// TIA Portal V19 export
TYPE "typePressureGuageRs485ControlNodeMonitoring"
TITLE = LBC_typeAnalogOutputControlNodeMonitoring
// Control Node Wapper monitoring values
// stored: Access Published
   STRUCT
      valid { ExternalAccessible := 'False'; ExternalVisible := 'False'; ExternalWritable := 'False'} : Bool;   // Manual mode parameters for axis control interface
      busy { ExternalAccessible := 'False'; ExternalVisible := 'False'; ExternalWritable := 'False'} : Bool;   // Manual mode parameters for axis control interface
      error { ExternalAccessible := 'False'; ExternalVisible := 'False'; ExternalWritable := 'False'} : Bool;   // Manual mode parameters for axis control interface
      status { ExternalAccessible := 'False'; ExternalVisible := 'False'; ExternalWritable := 'False'} : Word;   // 16#0000-16#7FFF: Status of the FB 16#8000-16#FFFF: Error identification (see following Table)
      limitHigh2 { ExternalAccessible := 'False'; ExternalVisible := 'False'; ExternalWritable := 'False'} : Bool;   // Manual mode parameters for axis control interface
      limitHigh1 { ExternalAccessible := 'False'; ExternalVisible := 'False'; ExternalWritable := 'False'} : Bool;   // Manual mode parameters for axis control interface
      limitLow1 { ExternalAccessible := 'False'; ExternalVisible := 'False'; ExternalWritable := 'False'} : Bool;   // Manual mode parameters for axis control interface
      limitLow2 { ExternalAccessible := 'False'; ExternalVisible := 'False'; ExternalWritable := 'False'} : Bool;   // Manual mode parameters for axis control interface
      maxValueReached { ExternalAccessible := 'False'; ExternalVisible := 'False'; ExternalWritable := 'False'} : Bool;   // Manual mode parameters for axis control interface
      minValueReached { ExternalAccessible := 'False'; ExternalVisible := 'False'; ExternalWritable := 'False'} : Bool;   // Manual mode parameters for axis control interface
   END_STRUCT;
END_TYPE
